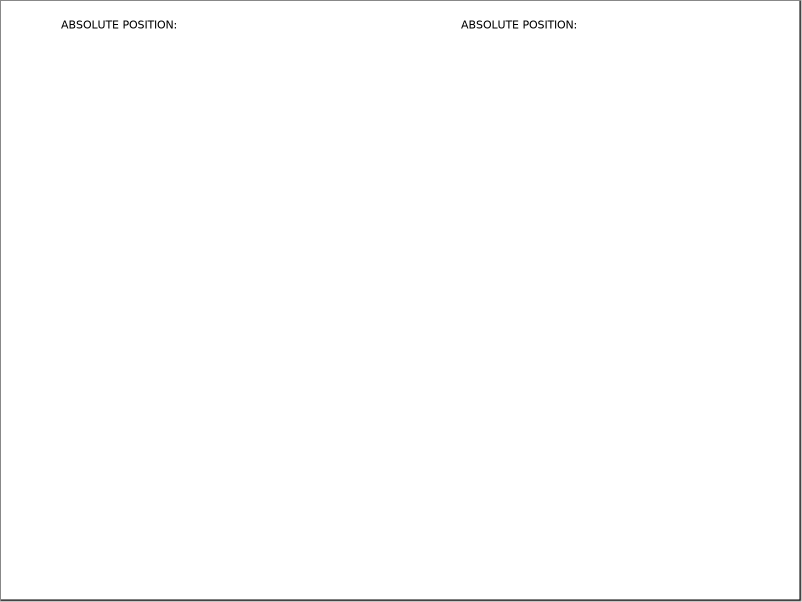
VISUALIZATION F34_Move_Continuous_Relative  // 802x602
    Rectangle (0,0 800x600)
    Label (10,10 170x30), "ABSOLUTE POSITION:"
    Label (410,10 170x30), "ABSOLUTE POSITION:"
END_VISUALIZATION

(* stored: Version 1.1.0.1, ProductVersion 3.1.4022.7
   Visu F34_Move_Continuous_Relative: Id {b7c9ed78-e61f-4b64-9366-53eb5d67f871} *)
